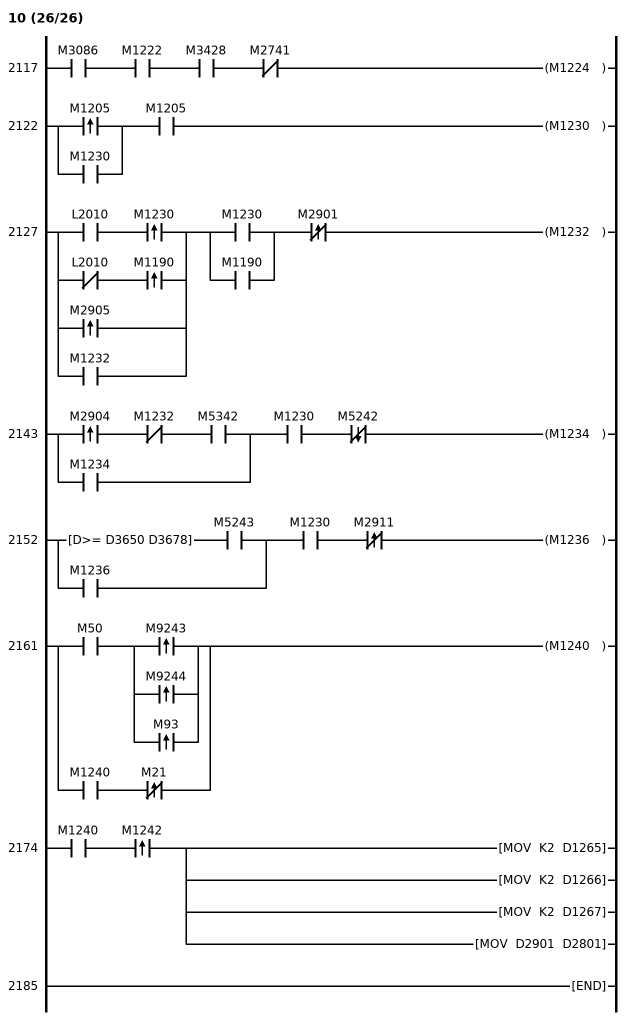
2117  LD      M3086
      AND     M1222
      AND     M3428
      ANI     M2741
      OUT     M1224
2122  LDP     M1205
      OR      M1230
      AND     M1205
      OUT     M1230
2127  LD      L2010
      ANDP    M1230
      LDI     L2010
      ANDP    M1190
      ORB
      ORP     M2905
      OR      M1232
      LD      M1230
      OR      M1190
      ANB
      ANDPI   M2901
      OUT     M1232
2143  LDP     M2904
      ANI     M1232
      AND     M5342
      OR      M1234
      AND     M1230
      ANDFI   M5242
      OUT     M1234
2152  LDD>=   D3650 D3678
      AND     M5243
      OR      M1236
      AND     M1230
      ANDPI   M2911
      OUT     M1236
2161  LD      M50
      LDP     M9243
      ORP     M9244
      ORP     M93
      ANB
      LD      M1240
      ANDPI   M21
      ORB
      OUT     M1240
2174  LD      M1240
      ANDP    M1242
      MOV     K2 D1265
      MOV     K2 D1266
      MOV     K2 D1267
      MOV     D2901 D2801
2185  END
END_PROGRAM

PROGRAM 20
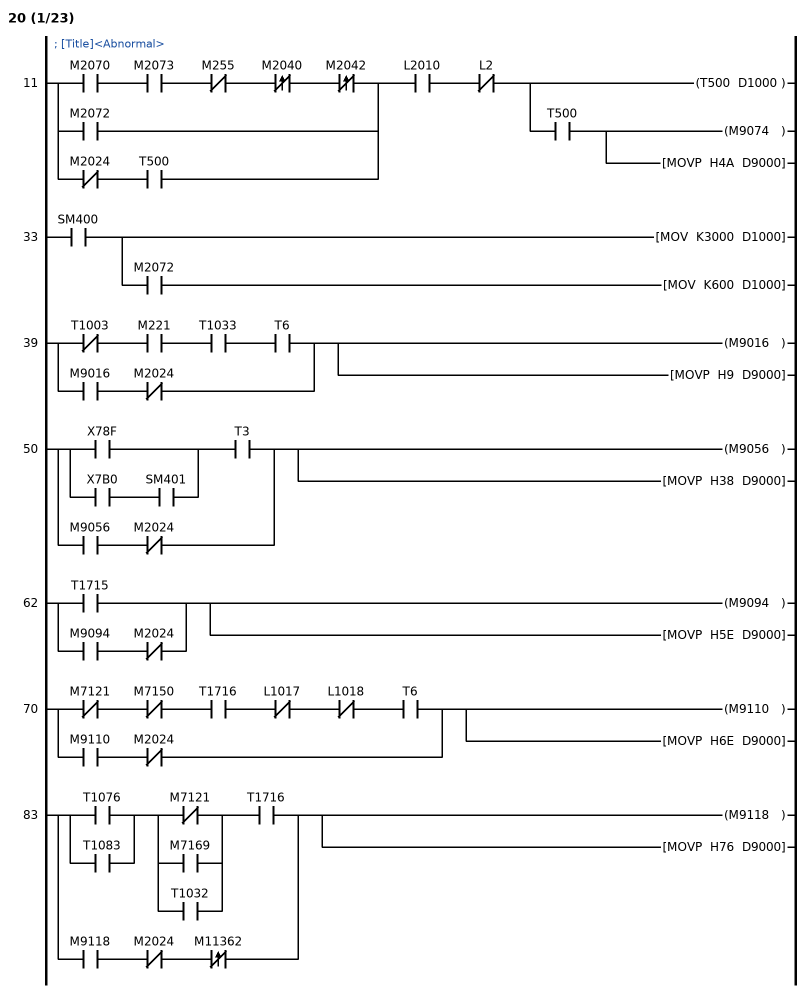
; [Title]<Abnormal>
11    LD      M2070
      AND     M2073
      ANI     M255
      ANDPI   M2040
      ANDPI   M2042
      OR      M2072
      LDI     M2024
      AND     T500
      ORB
      AND     L2010
      ANI     L2
      OUT     T500 D1000
      AND     T500
      OUT     M9074
      MOVP    H4A D9000
33    LD      SM400
      MOV     K3000 D1000
      AND     M2072
      MOV     K600 D1000
39    LDI     T1003
      AND     M221
      AND     T1033
      AND     T6
      LD      M9016
      ANI     M2024
      ORB
      OUT     M9016
      MOVP    H9 D9000
50    LD      X78F
      LD      X7B0
      AND     SM401
      ORB
      AND     T3
      LD      M9056
      ANI     M2024
      ORB
      OUT     M9056
      MOVP    H38 D9000
62    LD      T1715
      LD      M9094
      ANI     M2024
      ORB
      OUT     M9094
      MOVP    H5E D9000
70    LDI     M7121
      ANI     M7150
      AND     T1716
      ANI     L1017
      ANI     L1018
      AND     T6
      LD      M9110
      ANI     M2024
      ORB
      OUT     M9110
      MOVP    H6E D9000
83    LD      T1076
      OR      T1083
      LDI     M7121
      OR      M7169
      OR      T1032
      ANB
      AND     T1716
      LD      M9118
      ANI     M2024
      ANDPI   M11362
      ORB
      OUT     M9118
      MOVP    H76 D9000
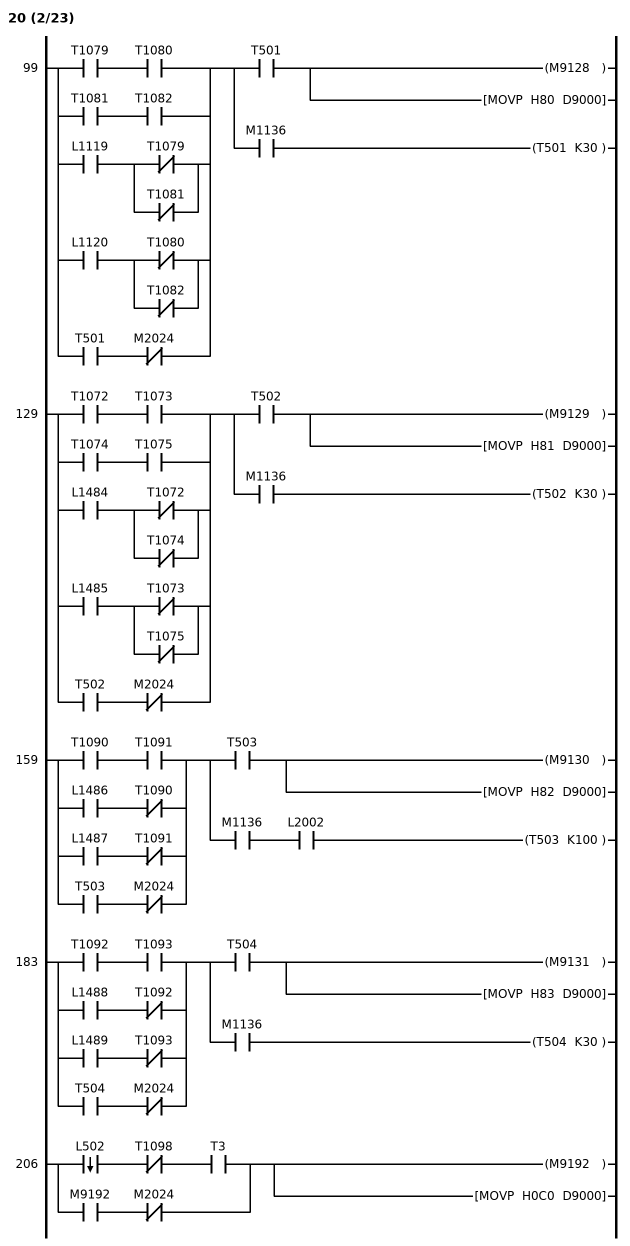
99    LD      T1079
      AND     T1080
      LD      T1081
      AND     T1082
      ORB
      LD      L1119
      LDI     T1079
      ORI     T1081
      ANB
      ORB
      LD      L1120
      LDI     T1080
      ORI     T1082
      ANB
      ORB
      LD      T501
      ANI     M2024
      ORB
      MPS
      AND     T501
      OUT     M9128
      MOVP    H80 D9000
      MPP
      AND     M1136
      OUT     T501 K30
129   LD      T1072
      AND     T1073
      LD      T1074
      AND     T1075
      ORB
      LD      L1484
      LDI     T1072
      ORI     T1074
      ANB
      ORB
      LD      L1485
      LDI     T1073
      ORI     T1075
      ANB
      ORB
      LD      T502
      ANI     M2024
      ORB
      MPS
      AND     T502
      OUT     M9129
      MOVP    H81 D9000
      MPP
      AND     M1136
      OUT     T502 K30
159   LD      T1090
      AND     T1091
      LD      L1486
      ANI     T1090
      ORB
      LD      L1487
      ANI     T1091
      ORB
      LD      T503
      ANI     M2024
      ORB
      MPS
      AND     T503
      OUT     M9130
      MOVP    H82 D9000
      MPP
      AND     M1136
      AND     L2002
      OUT     T503 K100
183   LD      T1092
      AND     T1093
      LD      L1488
      ANI     T1092
      ORB
      LD      L1489
      ANI     T1093
      ORB
      LD      T504
      ANI     M2024
      ORB
      MPS
      AND     T504
      OUT     M9131
      MOVP    H83 D9000
      MPP
      AND     M1136
      OUT     T504 K30
206   LDF     L502
      ANI     T1098
      AND     T3
      LD      M9192
      ANI     M2024
      ORB
      OUT     M9192
      MOVP    H0C0 D9000
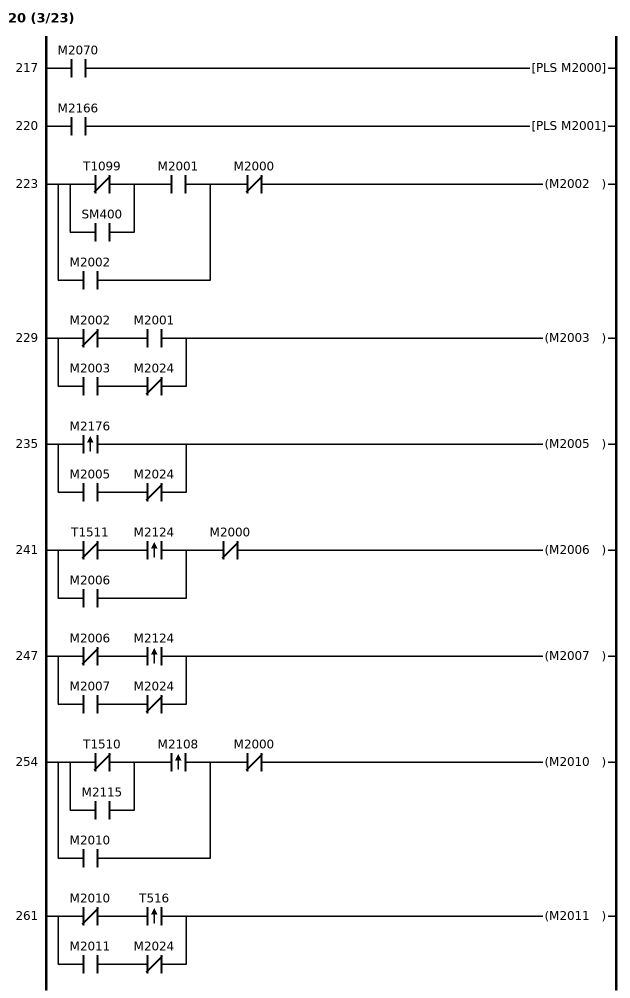
217   LD      M2070
      PLS     M2000
220   LD      M2166
      PLS     M2001
223   LDI     T1099
      OR      SM400
      AND     M2001
      OR      M2002
      ANI     M2000
      OUT     M2002
229   LDI     M2002
      AND     M2001
      LD      M2003
      ANI     M2024
      ORB
      OUT     M2003
235   LDP     M2176
      LD      M2005
      ANI     M2024
      ORB
      OUT     M2005
241   LDI     T1511
      ANDP    M2124
      OR      M2006
      ANI     M2000
      OUT     M2006
247   LDI     M2006
      ANDP    M2124
      LD      M2007
      ANI     M2024
      ORB
      OUT     M2007
254   LDI     T1510
      OR      M2115
      ANDP    M2108
      OR      M2010
      ANI     M2000
      OUT     M2010
261   LDI     M2010
      ANDP    T516
      LD      M2011
      ANI     M2024
      ORB
      OUT     M2011
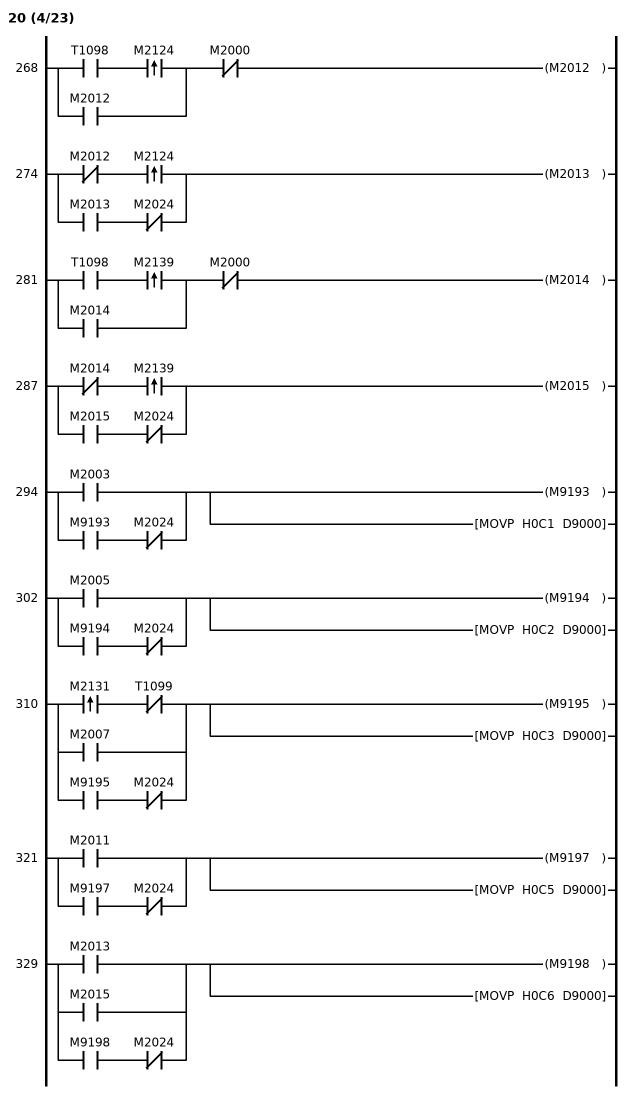
268   LD      T1098
      ANDP    M2124
      OR      M2012
      ANI     M2000
      OUT     M2012
274   LDI     M2012
      ANDP    M2124
      LD      M2013
      ANI     M2024
      ORB
      OUT     M2013
281   LD      T1098
      ANDP    M2139
      OR      M2014
      ANI     M2000
      OUT     M2014
287   LDI     M2014
      ANDP    M2139
      LD      M2015
      ANI     M2024
      ORB
      OUT     M2015
294   LD      M2003
      LD      M9193
      ANI     M2024
      ORB
      OUT     M9193
      MOVP    H0C1 D9000
302   LD      M2005
      LD      M9194
      ANI     M2024
      ORB
      OUT     M9194
      MOVP    H0C2 D9000
310   LDP     M2131
      ANI     T1099
      OR      M2007
      LD      M9195
      ANI     M2024
      ORB
      OUT     M9195
      MOVP    H0C3 D9000
321   LD      M2011
      LD      M9197
      ANI     M2024
      ORB
      OUT     M9197
      MOVP    H0C5 D9000
329   LD      M2013
      OR      M2015
      LD      M9198
      ANI     M2024
      ORB
      OUT     M9198
      MOVP    H0C6 D9000
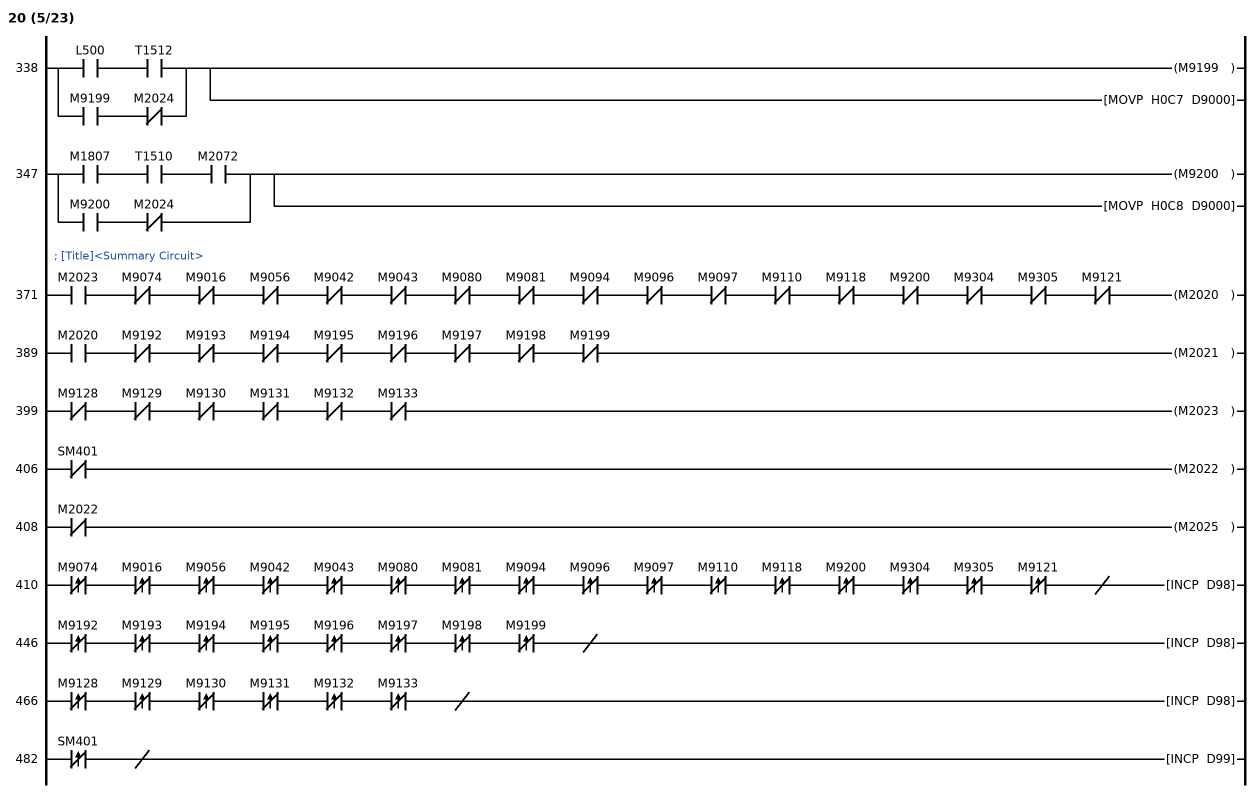
338   LD      L500
      AND     T1512
      LD      M9199
      ANI     M2024
      ORB
      OUT     M9199
      MOVP    H0C7 D9000
347   LD      M1807
      AND     T1510
      AND     M2072
      LD      M9200
      ANI     M2024
      ORB
      OUT     M9200
      MOVP    H0C8 D9000
; [Title]<Summary Circuit>
371   LD      M2023
      ANI     M9074
      ANI     M9016
      ANI     M9056
      ANI     M9042
      ANI     M9043
      ANI     M9080
      ANI     M9081
      ANI     M9094
      ANI     M9096
      ANI     M9097
      ANI     M9110
      ANI     M9118
      ANI     M9200
      ANI     M9304
      ANI     M9305
      ANI     M9121
      OUT     M2020
389   LD      M2020
      ANI     M9192
      ANI     M9193
      ANI     M9194
      ANI     M9195
      ANI     M9196
      ANI     M9197
      ANI     M9198
      ANI     M9199
      OUT     M2021
399   LDI     M9128
      ANI     M9129
      ANI     M9130
      ANI     M9131
      ANI     M9132
      ANI     M9133
      OUT     M2023
406   LDI     SM401
      OUT     M2022
408   LDI     M2022
      OUT     M2025
410   LDPI    M9074
      ANDPI   M9016
      ANDPI   M9056
      ANDPI   M9042
      ANDPI   M9043
      ANDPI   M9080
      ANDPI   M9081
      ANDPI   M9094
      ANDPI   M9096
      ANDPI   M9097
      ANDPI   M9110
      ANDPI   M9118
      ANDPI   M9200
      ANDPI   M9304
      ANDPI   M9305
      ANDPI   M9121
      INV
      INCP    D98
446   LDPI    M9192
      ANDPI   M9193
      ANDPI   M9194
      ANDPI   M9195
      ANDPI   M9196
      ANDPI   M9197
      ANDPI   M9198
      ANDPI   M9199
      INV
      INCP    D98
466   LDPI    M9128
      ANDPI   M9129
      ANDPI   M9130
      ANDPI   M9131
      ANDPI   M9132
      ANDPI   M9133
      INV
      INCP    D98
482   LDPI    SM401
      INV
      INCP    D99
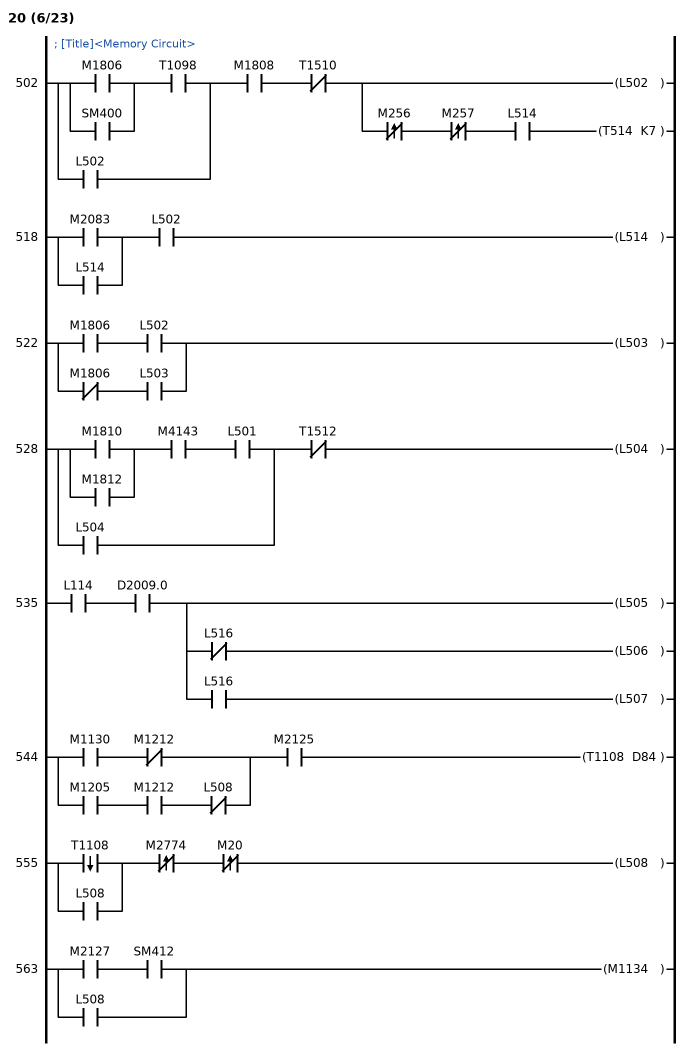
; [Title]<Memory Circuit>
502   LD      M1806
      OR      SM400
      AND     T1098
      OR      L502
      AND     M1808
      ANI     T1510
      OUT     L502
      ANDPI   M256
      ANDPI   M257
      AND     L514
      OUT     T514 K7
518   LD      M2083
      OR      L514
      AND     L502
      OUT     L514
522   LD      M1806
      AND     L502
      LDI     M1806
      AND     L503
      ORB
      OUT     L503
528   LD      M1810
      OR      M1812
      AND     M4143
      AND     L501
      OR      L504
      ANI     T1512
      OUT     L504
535   LD      L114
      AND     D2009.0
      OUT     L505
      MPS
      ANI     L516
      OUT     L506
      MPP
      AND     L516
      OUT     L507
544   LD      M1130
      ANI     M1212
      LD      M1205
      AND     M1212
      ANI     L508
      ORB
      AND     M2125
      OUT     T1108 D84
555   LDF     T1108
      OR      L508
      ANDPI   M2774
      ANDPI   M20
      OUT     L508
563   LD      M2127
      AND     SM412
      OR      L508
      OUT     M1134
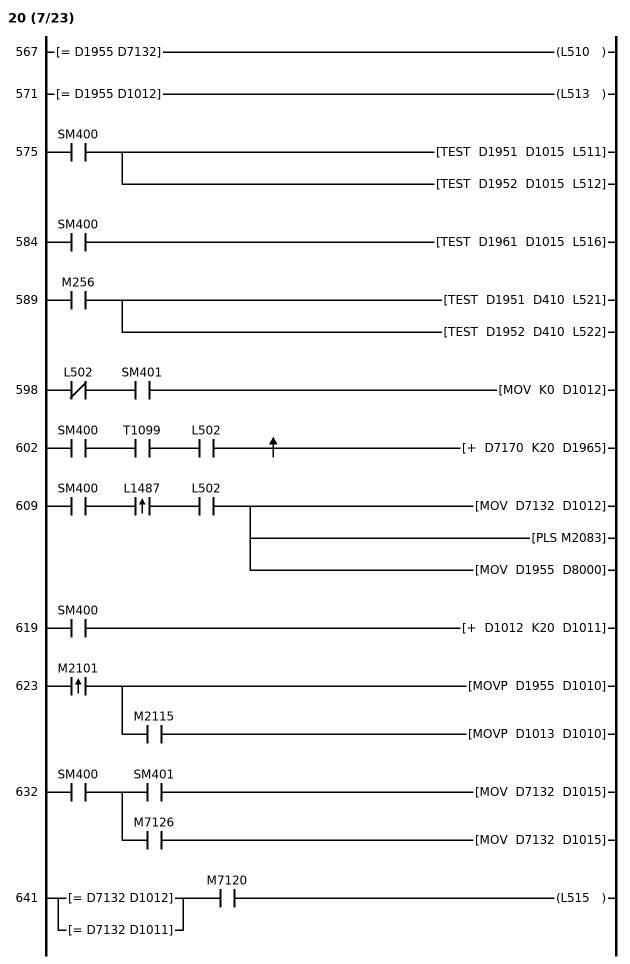
567   LD=     D1955 D7132
      OUT     L510
571   LD=     D1955 D1012
      OUT     L513
575   LD      SM400
      TEST    D1951 D1015 L511
      TEST    D1952 D1015 L512
584   LD      SM400
      TEST    D1961 D1015 L516
589   LD      M256
      TEST    D1951 D410 L521
      TEST    D1952 D410 L522
598   LDI     L502
      AND     SM401
      MOV     K0 D1012
602   LD      SM400
      AND     T1099
      AND     L502
      MEP
      +       D7170 K20 D1965
609   LD      SM400
      ANDP    L1487
      AND     L502
      MOV     D7132 D1012
      PLS     M2083
      MOV     D1955 D8000
619   LD      SM400
      +       D1012 K20 D1011
623   LDP     M2101
      MOVP    D1955 D1010
      AND     M2115
      MOVP    D1013 D1010
632   LD      SM400
      MPS
      AND     SM401
      MOV     D7132 D1015
      MPP
      AND     M7126
      MOV     D7132 D1015
641   LD=     D7132 D1012
      OR=     D7132 D1011
      AND     M7120
      OUT     L515
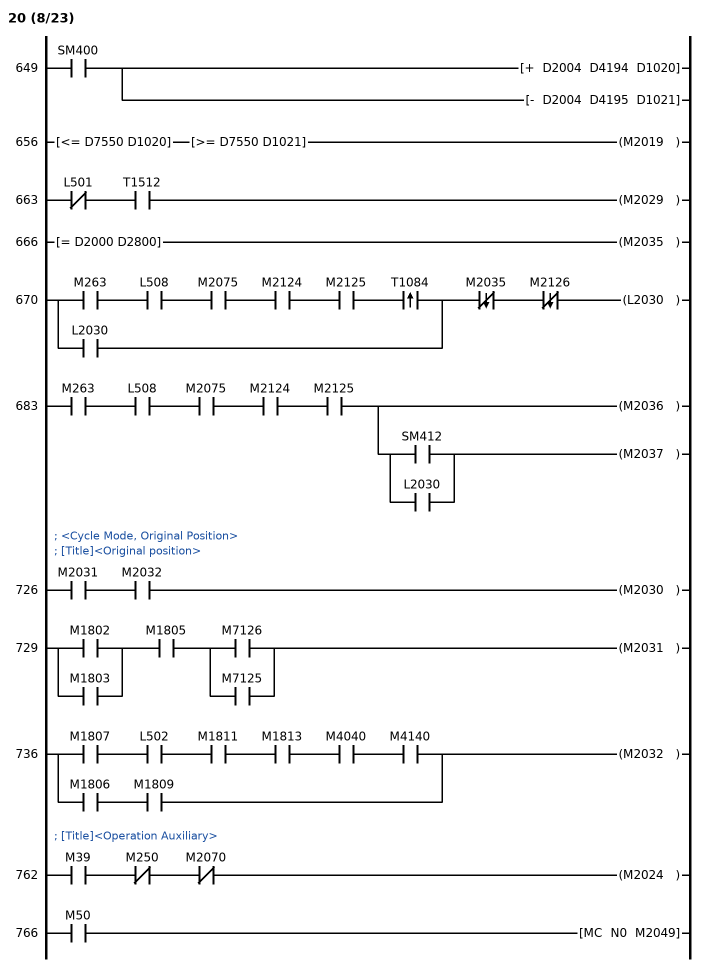
649   LD      SM400
      +       D2004 D4194 D1020
      -       D2004 D4195 D1021
656   LD<=    D7550 D1020
      AND>=   D7550 D1021
      OUT     M2019
663   LDI     L501
      AND     T1512
      OUT     M2029
666   LD=     D2000 D2800
      OUT     M2035
670   LD      M263
      AND     L508
      AND     M2075
      AND     M2124
      AND     M2125
      ANDP    T1084
      OR      L2030
      ANDFI   M2035
      ANDFI   M2126
      OUT     L2030
683   LD      M263
      AND     L508
      AND     M2075
      AND     M2124
      AND     M2125
      OUT     M2036
      LD      SM412
      OR      L2030
      ANB
      OUT     M2037
; <Cycle Mode, Original Position>
; [Title]<Original position>
726   LD      M2031
      AND     M2032
      OUT     M2030
729   LD      M1802
      OR      M1803
      AND     M1805
      LD      M7126
      OR      M7125
      ANB
      OUT     M2031
736   LD      M1807
      AND     L502
      AND     M1811
      AND     M1813
      AND     M4040
      AND     M4140
      LD      M1806
      AND     M1809
      ORB
      OUT     M2032
; [Title]<Operation Auxiliary>
762   LD      M39
      ANI     M250
      ANI     M2070
      OUT     M2024
766   LD      M50
      MC      N0 M2049
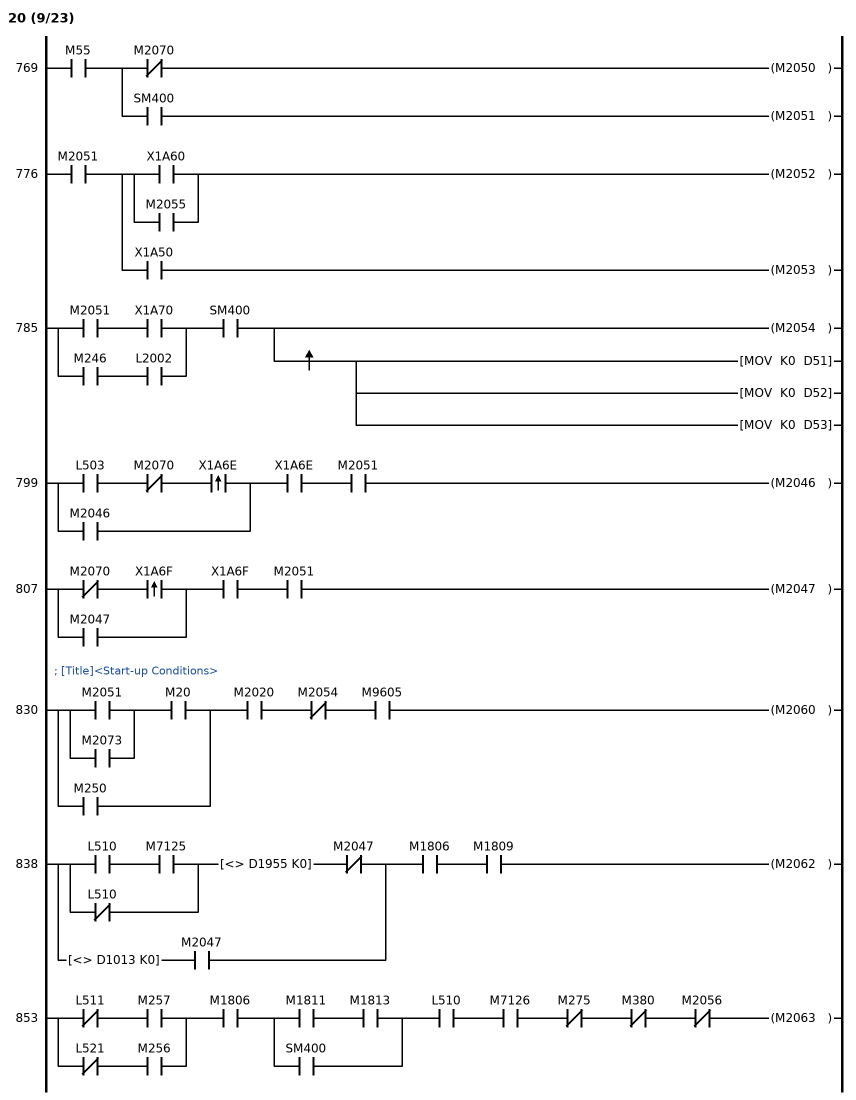
769   LD      M55
      MPS
      ANI     M2070
      OUT     M2050
      MPP
      AND     SM400
      OUT     M2051
776   LD      M2051
      MPS
      LD      X1A60
      OR      M2055
      ANB
      OUT     M2052
      MPP
      AND     X1A50
      OUT     M2053
785   LD      M2051
      AND     X1A70
      LD      M246
      AND     L2002
      ORB
      AND     SM400
      OUT     M2054
      MEP
      MOV     K0 D51
      MOV     K0 D52
      MOV     K0 D53
799   LD      L503
      ANI     M2070
      ANDP    X1A6E
      OR      M2046
      AND     X1A6E
      AND     M2051
      OUT     M2046
807   LDI     M2070
      ANDP    X1A6F
      OR      M2047
      AND     X1A6F
      AND     M2051
      OUT     M2047
; [Title]<Start-up Conditions>
830   LD      M2051
      OR      M2073
      AND     M20
      OR      M250
      AND     M2020
      ANI     M2054
      AND     M9605
      OUT     M2060
838   LD      L510
      AND     M7125
      ORI     L510
      AND<>   D1955 K0
      ANI     M2047
      LD<>    D1013 K0
      AND     M2047
      ORB
      AND     M1806
      AND     M1809
      OUT     M2062
853   LDI     L511
      AND     M257
      LDI     L521
      AND     M256
      ORB
      AND     M1806
      LD      M1811
      AND     M1813
      OR      SM400
      ANB
      AND     L510
      AND     M7126
      ANI     M275
      ANI     M380
      ANI     M2056
      OUT     M2063
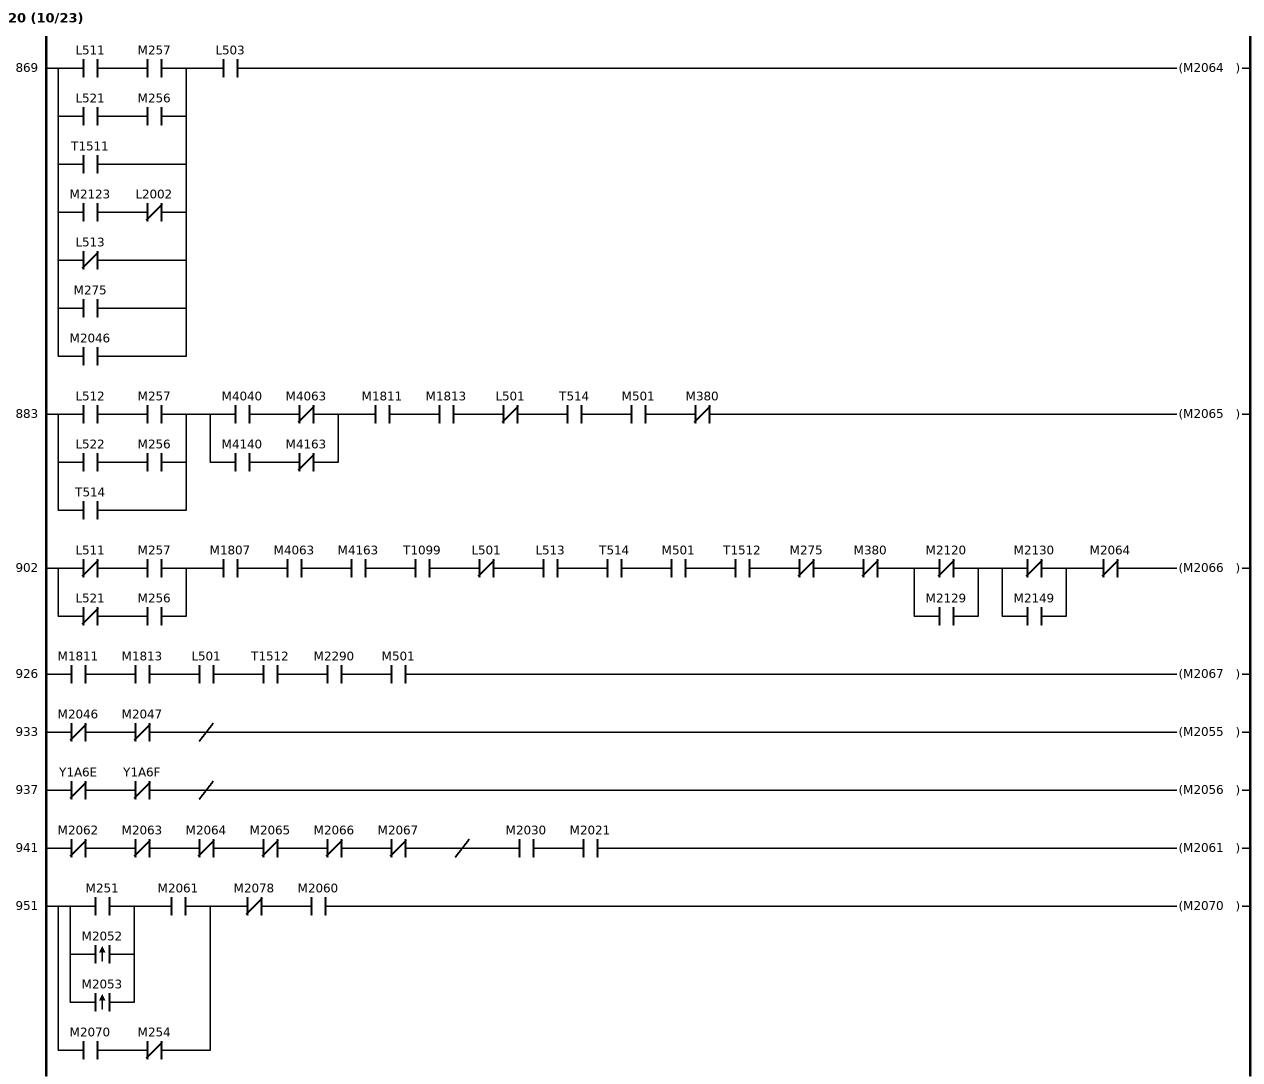
869   LD      L511
      AND     M257
      LD      L521
      AND     M256
      ORB
      OR      T1511
      LD      M2123
      ANI     L2002
      ORB
      ORI     L513
      OR      M275
      OR      M2046
      AND     L503
      OUT     M2064
883   LD      L512
      AND     M257
      LD      L522
      AND     M256
      ORB
      OR      T514
      LD      M4040
      ANI     M4063
      LD      M4140
      ANI     M4163
      ORB
      ANB
      AND     M1811
      AND     M1813
      ANI     L501
      AND     T514
      AND     M501
      ANI     M380
      OUT     M2065
902   LDI     L511
      AND     M257
      LDI     L521
      AND     M256
      ORB
      AND     M1807
      AND     M4063
      AND     M4163
      AND     T1099
      ANI     L501
      AND     L513
      AND     T514
      AND     M501
      AND     T1512
      ANI     M275
      ANI     M380
      LDI     M2120
      OR      M2129
      ANB
      LDI     M2130
      OR      M2149
      ANB
      ANI     M2064
      OUT     M2066
926   LD      M1811
      AND     M1813
      AND     L501
      AND     T1512
      AND     M2290
      AND     M501
      OUT     M2067
933   LDI     M2046
      ANI     M2047
      INV
      OUT     M2055
937   LDI     Y1A6E
      ANI     Y1A6F
      INV
      OUT     M2056
941   LDI     M2062
      ANI     M2063
      ANI     M2064
      ANI     M2065
      ANI     M2066
      ANI     M2067
      INV
      AND     M2030
      AND     M2021
      OUT     M2061
951   LD      M251
      ORP     M2052
      ORP     M2053
      AND     M2061
      LD      M2070
      ANI     M254
      ORB
      ANI     M2078
      AND     M2060
      OUT     M2070
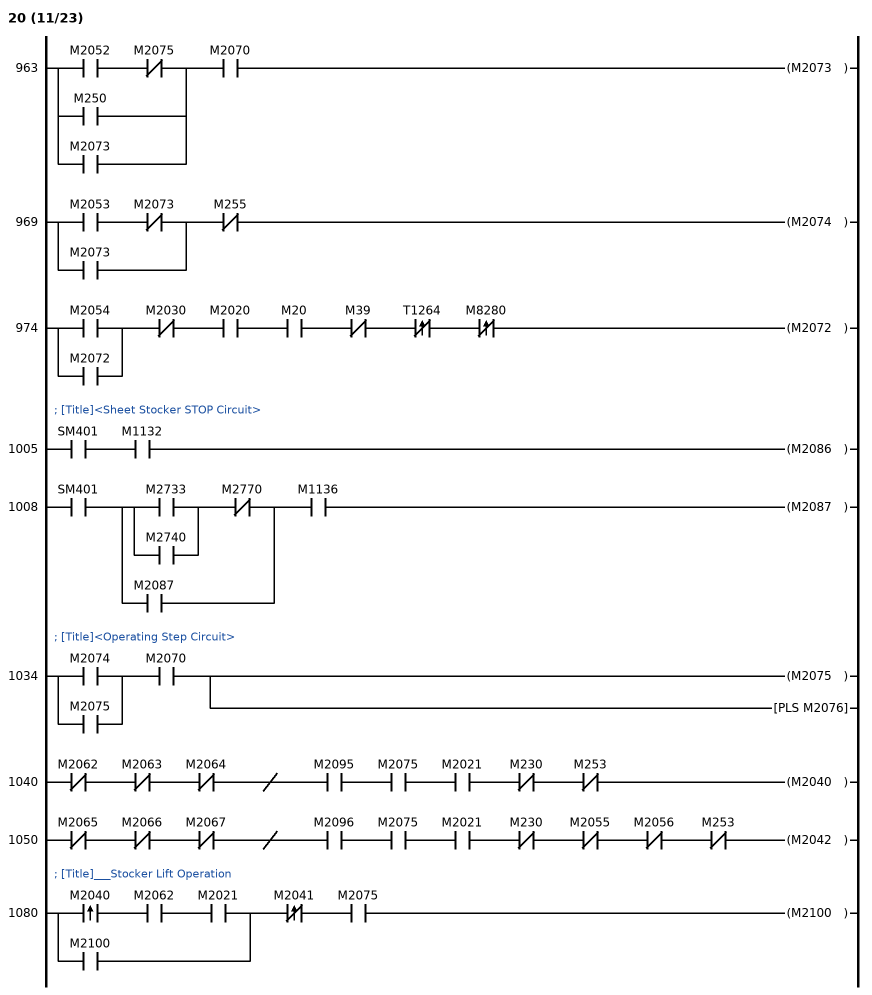
963   LD      M2052
      ANI     M2075
      OR      M250
      OR      M2073
      AND     M2070
      OUT     M2073
969   LD      M2053
      ANI     M2073
      OR      M2073
      ANI     M255
      OUT     M2074
974   LD      M2054
      OR      M2072
      ANI     M2030
      AND     M2020
      AND     M20
      ANI     M39
      ANDPI   T1264
      ANDPI   M8280
      OUT     M2072
; [Title]<Sheet Stocker STOP Circuit>
1005  LD      SM401
      AND     M1132
      OUT     M2086
1008  LD      SM401
      LD      M2733
      OR      M2740
      ANI     M2770
      OR      M2087
      ANB
      AND     M1136
      OUT     M2087
; [Title]<Operating Step Circuit>
1034  LD      M2074
      OR      M2075
      AND     M2070
      OUT     M2075
      PLS     M2076
1040  LDI     M2062
      ANI     M2063
      ANI     M2064
      INV
      AND     M2095
      AND     M2075
      AND     M2021
      ANI     M230
      ANI     M253
      OUT     M2040
1050  LDI     M2065
      ANI     M2066
      ANI     M2067
      INV
      AND     M2096
      AND     M2075
      AND     M2021
      ANI     M230
      ANI     M2055
      ANI     M2056
      ANI     M253
      OUT     M2042
; [Title]___Stocker Lift Operation
1080  LDP     M2040
      AND     M2062
      AND     M2021
      OR      M2100
      ANDPI   M2041
      AND     M2075
      OUT     M2100
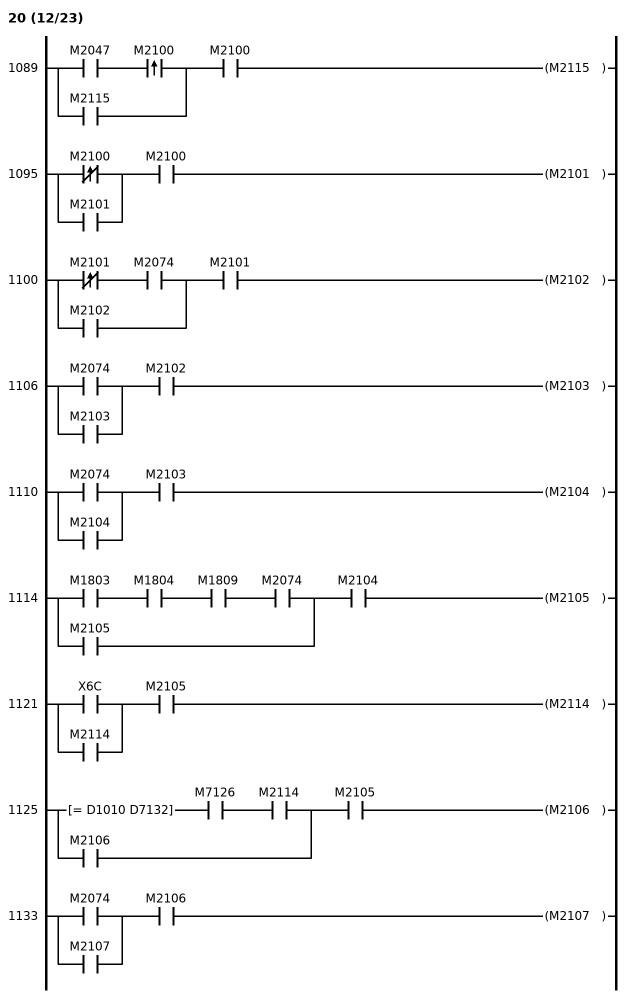
1089  LD      M2047
      ANDP    M2100
      OR      M2115
      AND     M2100
      OUT     M2115
1095  LDPI    M2100
      OR      M2101
      AND     M2100
      OUT     M2101
1100  LDPI    M2101
      AND     M2074
      OR      M2102
      AND     M2101
      OUT     M2102
1106  LD      M2074
      OR      M2103
      AND     M2102
      OUT     M2103
1110  LD      M2074
      OR      M2104
      AND     M2103
      OUT     M2104
1114  LD      M1803
      AND     M1804
      AND     M1809
      AND     M2074
      OR      M2105
      AND     M2104
      OUT     M2105
1121  LD      X6C
      OR      M2114
      AND     M2105
      OUT     M2114
1125  LD=     D1010 D7132
      AND     M7126
      AND     M2114
      OR      M2106
      AND     M2105
      OUT     M2106
1133  LD      M2074
      OR      M2107
      AND     M2106
      OUT     M2107
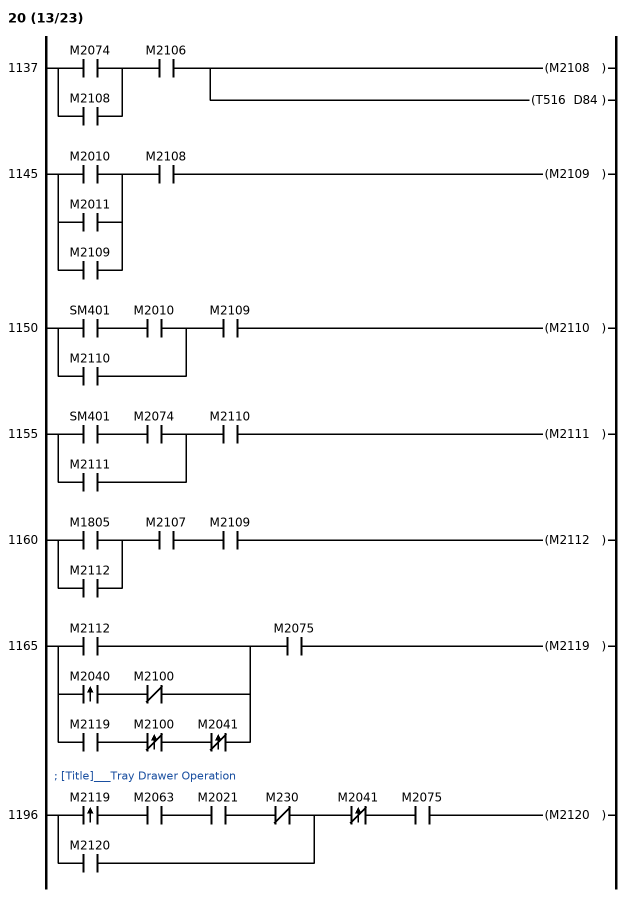
1137  LD      M2074
      OR      M2108
      AND     M2106
      OUT     M2108
      OUT     T516 D84
1145  LD      M2010
      OR      M2011
      OR      M2109
      AND     M2108
      OUT     M2109
1150  LD      SM401
      AND     M2010
      OR      M2110
      AND     M2109
      OUT     M2110
1155  LD      SM401
      AND     M2074
      OR      M2111
      AND     M2110
      OUT     M2111
1160  LD      M1805
      OR      M2112
      AND     M2107
      AND     M2109
      OUT     M2112
1165  LD      M2112
      LDP     M2040
      ANI     M2100
      ORB
      LD      M2119
      ANDPI   M2100
      ANDPI   M2041
      ORB
      AND     M2075
      OUT     M2119
; [Title]___Tray Drawer Operation
1196  LDP     M2119
      AND     M2063
      AND     M2021
      ANI     M230
      OR      M2120
      ANDPI   M2041
      AND     M2075
      OUT     M2120
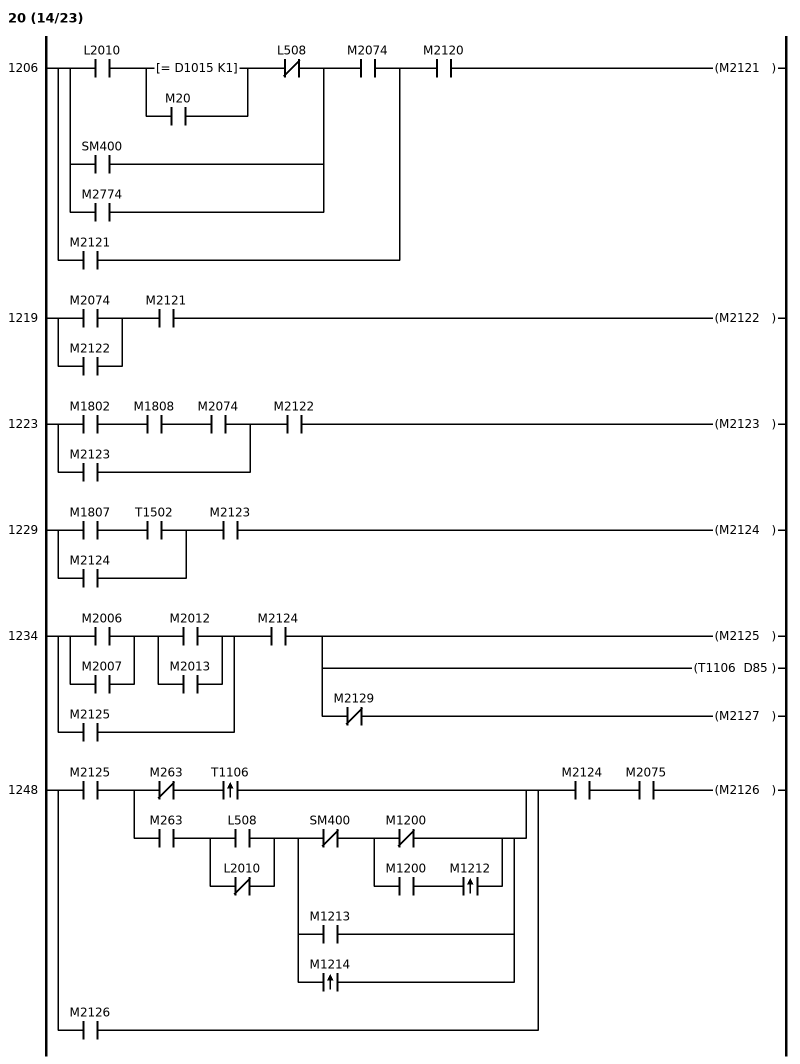
1206  LD      L2010
      LD=     D1015 K1
      OR      M20
      ANB
      ANI     L508
      OR      SM400
      OR      M2774
      AND     M2074
      OR      M2121
      AND     M2120
      OUT     M2121
1219  LD      M2074
      OR      M2122
      AND     M2121
      OUT     M2122
1223  LD      M1802
      AND     M1808
      AND     M2074
      OR      M2123
      AND     M2122
      OUT     M2123
1229  LD      M1807
      AND     T1502
      OR      M2124
      AND     M2123
      OUT     M2124
1234  LD      M2006
      OR      M2007
      LD      M2012
      OR      M2013
      ANB
      OR      M2125
      AND     M2124
      OUT     M2125
      OUT     T1106 D85
      ANI     M2129
      OUT     M2127
1248  LD      M2125
      LDI     M263
      ANDP    T1106
      LD      M263
      LD      L508
      ORI     L2010
      ANB
      LDI     SM400
      LDI     M1200
      LD      M1200
      ANDP    M1212
      ORB
      ANB
      OR      M1213
      ORP     M1214
      ANB
      ORB
      ANB
      OR      M2126
      AND     M2124
      AND     M2075
      OUT     M2126
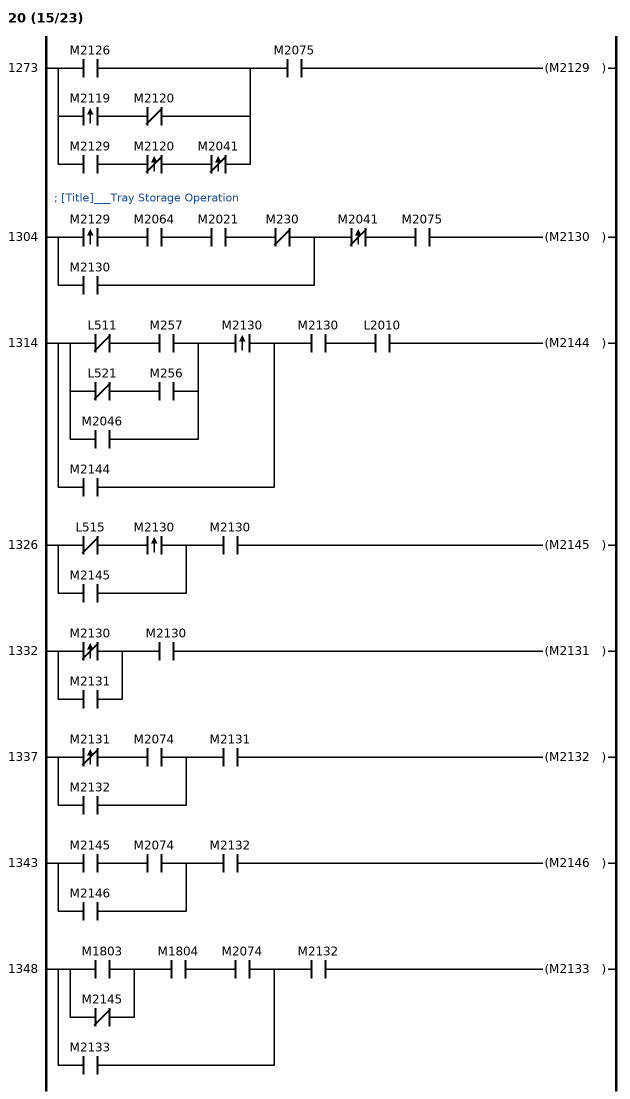
1273  LD      M2126
      LDP     M2119
      ANI     M2120
      ORB
      LD      M2129
      ANDPI   M2120
      ANDPI   M2041
      ORB
      AND     M2075
      OUT     M2129
; [Title]___Tray Storage Operation
1304  LDP     M2129
      AND     M2064
      AND     M2021
      ANI     M230
      OR      M2130
      ANDPI   M2041
      AND     M2075
      OUT     M2130
1314  LDI     L511
      AND     M257
      LDI     L521
      AND     M256
      ORB
      OR      M2046
      ANDP    M2130
      OR      M2144
      AND     M2130
      AND     L2010
      OUT     M2144
1326  LDI     L515
      ANDP    M2130
      OR      M2145
      AND     M2130
      OUT     M2145
1332  LDPI    M2130
      OR      M2131
      AND     M2130
      OUT     M2131
1337  LDPI    M2131
      AND     M2074
      OR      M2132
      AND     M2131
      OUT     M2132
1343  LD      M2145
      AND     M2074
      OR      M2146
      AND     M2132
      OUT     M2146
1348  LD      M1803
      ORI     M2145
      AND     M1804
      AND     M2074
      OR      M2133
      AND     M2132
      OUT     M2133
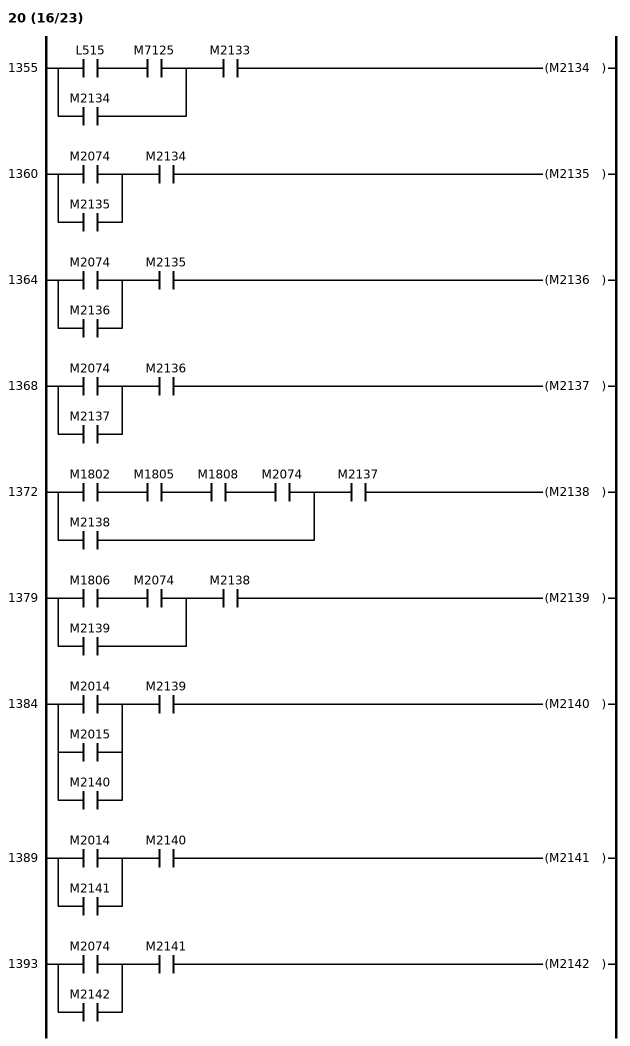
1355  LD      L515
      AND     M7125
      OR      M2134
      AND     M2133
      OUT     M2134
1360  LD      M2074
      OR      M2135
      AND     M2134
      OUT     M2135
1364  LD      M2074
      OR      M2136
      AND     M2135
      OUT     M2136
1368  LD      M2074
      OR      M2137
      AND     M2136
      OUT     M2137
1372  LD      M1802
      AND     M1805
      AND     M1808
      AND     M2074
      OR      M2138
      AND     M2137
      OUT     M2138
1379  LD      M1806
      AND     M2074
      OR      M2139
      AND     M2138
      OUT     M2139
1384  LD      M2014
      OR      M2015
      OR      M2140
      AND     M2139
      OUT     M2140
1389  LD      M2014
      OR      M2141
      AND     M2140
      OUT     M2141
1393  LD      M2074
      OR      M2142
      AND     M2141
      OUT     M2142
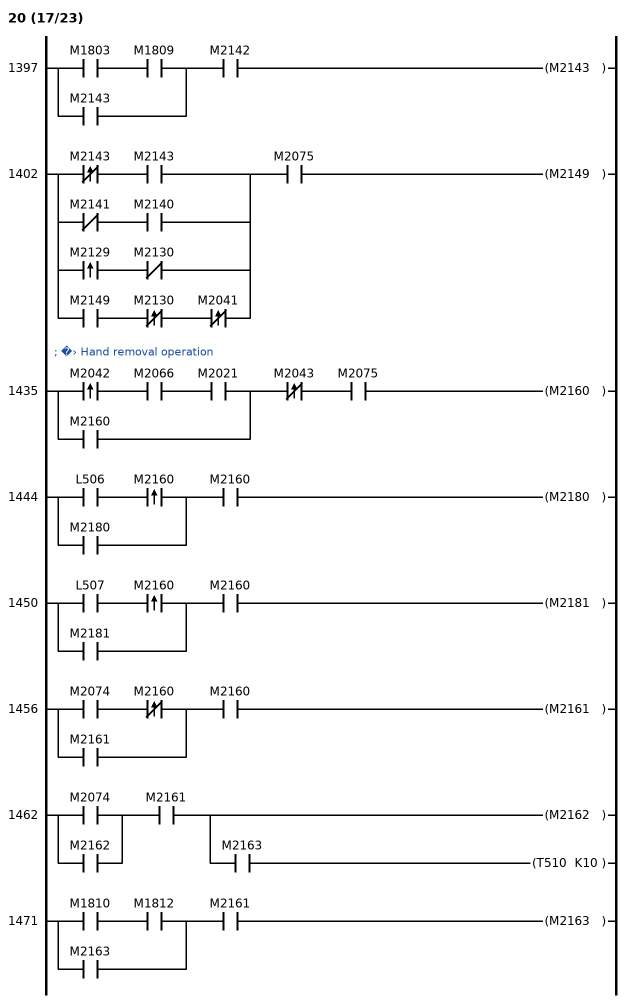
1397  LD      M1803
      AND     M1809
      OR      M2143
      AND     M2142
      OUT     M2143
1402  LDPI    M2143
      AND     M2143
      LDI     M2141
      AND     M2140
      ORB
      LDP     M2129
      ANI     M2130
      ORB
      LD      M2149
      ANDPI   M2130
      ANDPI   M2041
      ORB
      AND     M2075
      OUT     M2149
; �› Hand removal operation
1435  LDP     M2042
      AND     M2066
      AND     M2021
      OR      M2160
      ANDPI   M2043
      AND     M2075
      OUT     M2160
1444  LD      L506
      ANDP    M2160
      OR      M2180
      AND     M2160
      OUT     M2180
1450  LD      L507
      ANDP    M2160
      OR      M2181
      AND     M2160
      OUT     M2181
1456  LD      M2074
      ANDPI   M2160
      OR      M2161
      AND     M2160
      OUT     M2161
1462  LD      M2074
      OR      M2162
      AND     M2161
      OUT     M2162
      AND     M2163
      OUT     T510 K10
1471  LD      M1810
      AND     M1812
      OR      M2163
      AND     M2161
      OUT     M2163
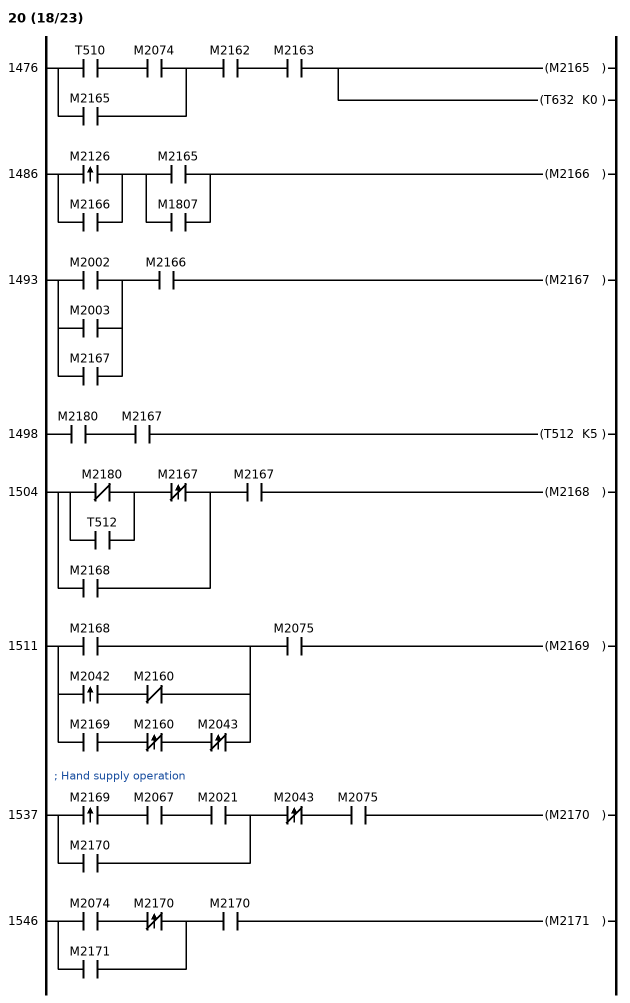
1476  LD      T510
      AND     M2074
      OR      M2165
      AND     M2162
      AND     M2163
      OUT     M2165
      OUT     T632 K0
1486  LDP     M2126
      OR      M2166
      LD      M2165
      OR      M1807
      ANB
      OUT     M2166
1493  LD      M2002
      OR      M2003
      OR      M2167
      AND     M2166
      OUT     M2167
1498  LD      M2180
      AND     M2167
      OUT     T512 K5
1504  LDI     M2180
      OR      T512
      ANDPI   M2167
      OR      M2168
      AND     M2167
      OUT     M2168
1511  LD      M2168
      LDP     M2042
      ANI     M2160
      ORB
      LD      M2169
      ANDPI   M2160
      ANDPI   M2043
      ORB
      AND     M2075
      OUT     M2169
; Hand supply operation
1537  LDP     M2169
      AND     M2067
      AND     M2021
      OR      M2170
      ANDPI   M2043
      AND     M2075
      OUT     M2170
1546  LD      M2074
      ANDPI   M2170
      OR      M2171
      AND     M2170
      OUT     M2171
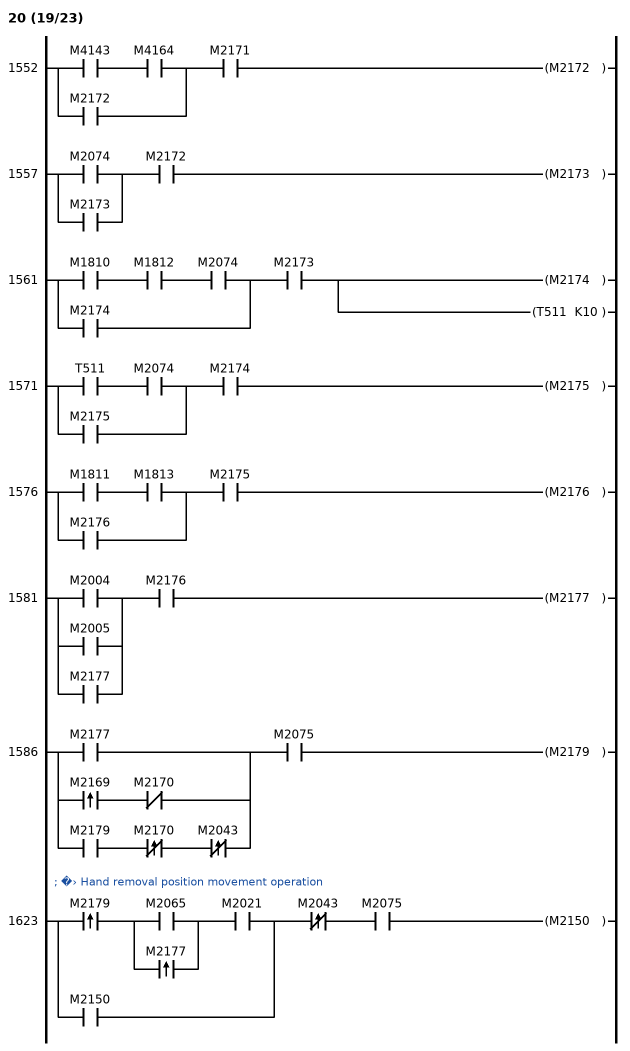
1552  LD      M4143
      AND     M4164
      OR      M2172
      AND     M2171
      OUT     M2172
1557  LD      M2074
      OR      M2173
      AND     M2172
      OUT     M2173
1561  LD      M1810
      AND     M1812
      AND     M2074
      OR      M2174
      AND     M2173
      OUT     M2174
      OUT     T511 K10
1571  LD      T511
      AND     M2074
      OR      M2175
      AND     M2174
      OUT     M2175
1576  LD      M1811
      AND     M1813
      OR      M2176
      AND     M2175
      OUT     M2176
1581  LD      M2004
      OR      M2005
      OR      M2177
      AND     M2176
      OUT     M2177
1586  LD      M2177
      LDP     M2169
      ANI     M2170
      ORB
      LD      M2179
      ANDPI   M2170
      ANDPI   M2043
      ORB
      AND     M2075
      OUT     M2179
; �› Hand removal position movement operation
1623  LDP     M2179
      LD      M2065
      ORP     M2177
      ANB
      AND     M2021
      OR      M2150
      ANDPI   M2043
      AND     M2075
      OUT     M2150
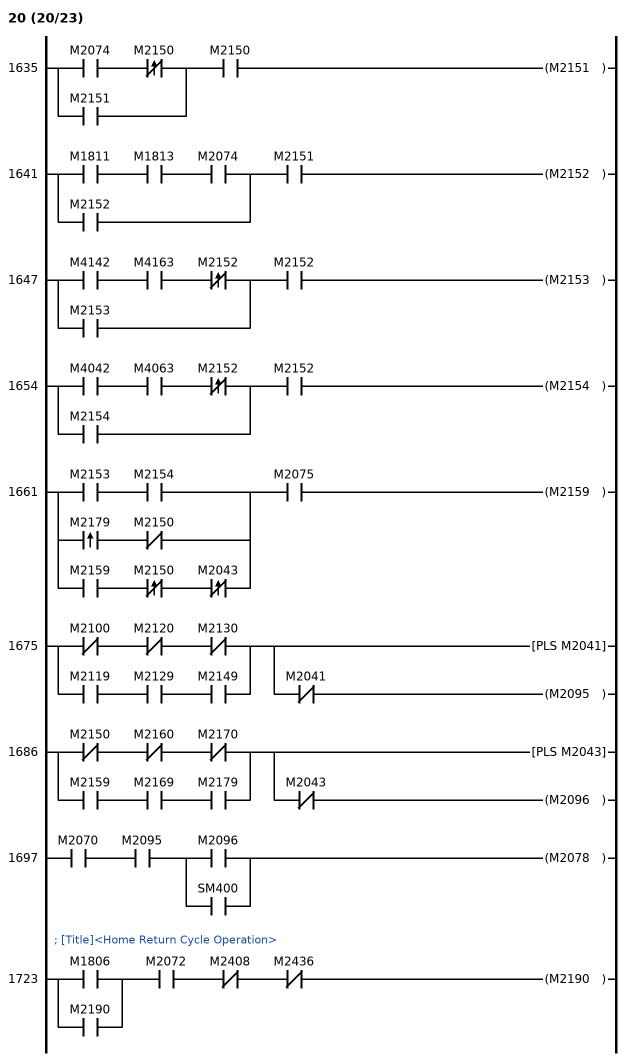
1635  LD      M2074
      ANDPI   M2150
      OR      M2151
      AND     M2150
      OUT     M2151
1641  LD      M1811
      AND     M1813
      AND     M2074
      OR      M2152
      AND     M2151
      OUT     M2152
1647  LD      M4142
      AND     M4163
      ANDPI   M2152
      OR      M2153
      AND     M2152
      OUT     M2153
1654  LD      M4042
      AND     M4063
      ANDPI   M2152
      OR      M2154
      AND     M2152
      OUT     M2154
1661  LD      M2153
      AND     M2154
      LDP     M2179
      ANI     M2150
      ORB
      LD      M2159
      ANDPI   M2150
      ANDPI   M2043
      ORB
      AND     M2075
      OUT     M2159
1675  LDI     M2100
      ANI     M2120
      ANI     M2130
      LD      M2119
      AND     M2129
      AND     M2149
      ORB
      PLS     M2041
      ANI     M2041
      OUT     M2095
1686  LDI     M2150
      ANI     M2160
      ANI     M2170
      LD      M2159
      AND     M2169
      AND     M2179
      ORB
      PLS     M2043
      ANI     M2043
      OUT     M2096
1697  LD      M2070
      AND     M2095
      LD      M2096
      OR      SM400
      ANB
      OUT     M2078
; [Title]<Home Return Cycle Operation>
1723  LD      M1806
      OR      M2190
      AND     M2072
      ANI     M2408
      ANI     M2436
      OUT     M2190
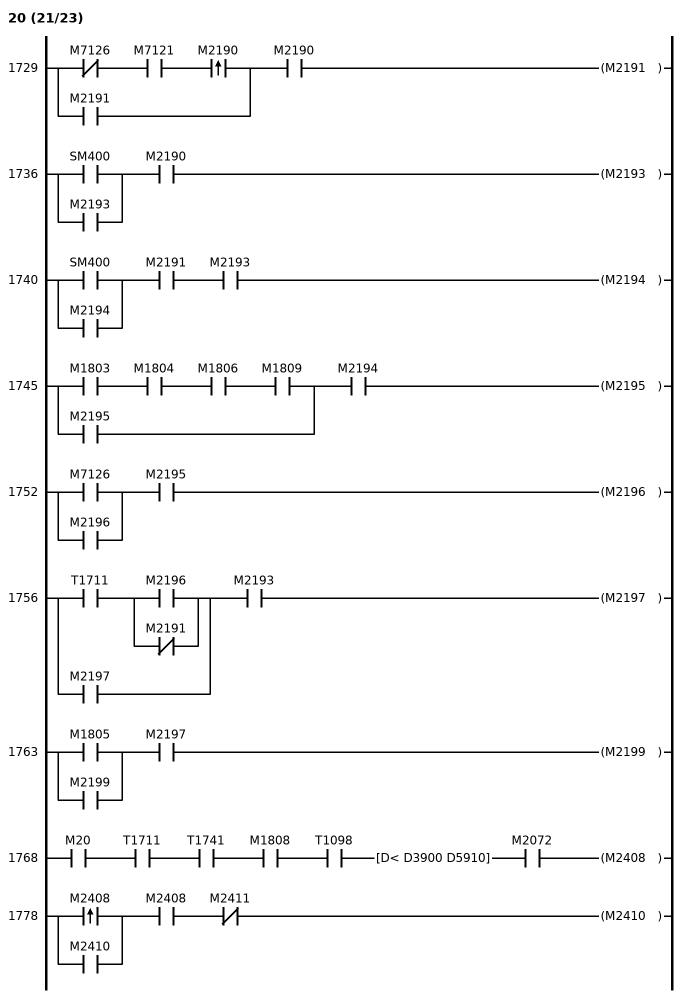
1729  LDI     M7126
      AND     M7121
      ANDP    M2190
      OR      M2191
      AND     M2190
      OUT     M2191
1736  LD      SM400
      OR      M2193
      AND     M2190
      OUT     M2193
1740  LD      SM400
      OR      M2194
      AND     M2191
      AND     M2193
      OUT     M2194
1745  LD      M1803
      AND     M1804
      AND     M1806
      AND     M1809
      OR      M2195
      AND     M2194
      OUT     M2195
1752  LD      M7126
      OR      M2196
      AND     M2195
      OUT     M2196
1756  LD      T1711
      LD      M2196
      ORI     M2191
      ANB
      OR      M2197
      AND     M2193
      OUT     M2197
1763  LD      M1805
      OR      M2199
      AND     M2197
      OUT     M2199
; 
1768  LD      M20
      AND     T1711
      AND     T1741
      AND     M1808
      AND     T1098
      ANDD<   D3900 D5910
      AND     M2072
      OUT     M2408
1778  LDP     M2408
      OR      M2410
      AND     M2408
      ANI     M2411
      OUT     M2410
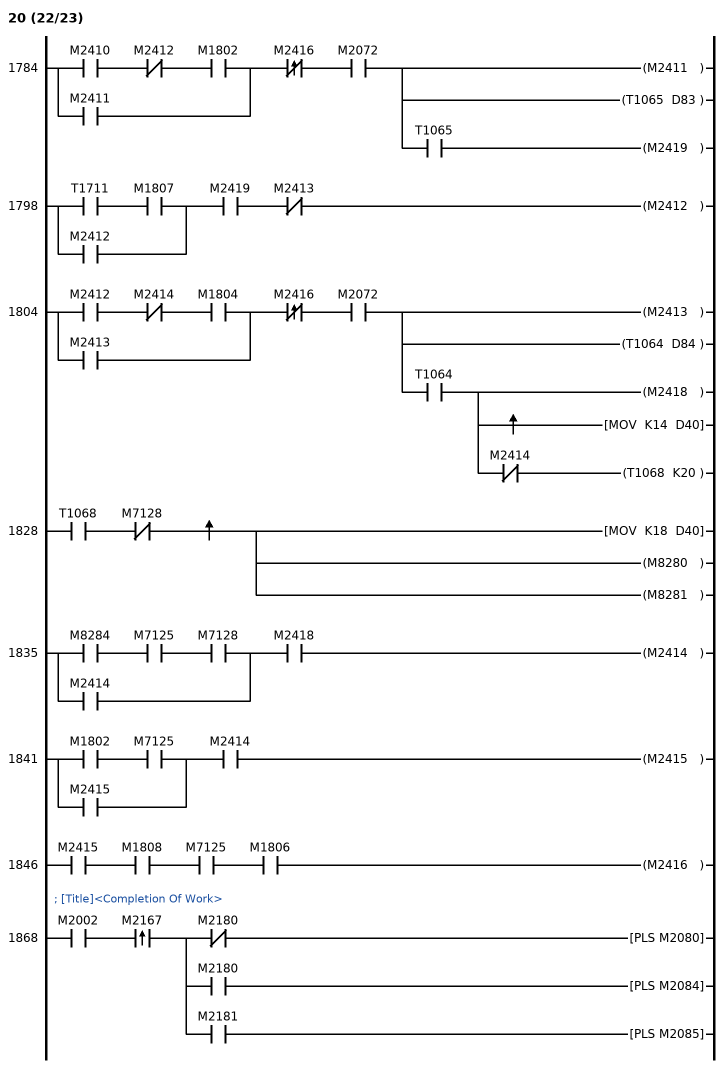
1784  LD      M2410
      ANI     M2412
      AND     M1802
      OR      M2411
      ANDPI   M2416
      AND     M2072
      OUT     M2411
      OUT     T1065 D83
      AND     T1065
      OUT     M2419
1798  LD      T1711
      AND     M1807
      OR      M2412
      AND     M2419
      ANI     M2413
      OUT     M2412
1804  LD      M2412
      ANI     M2414
      AND     M1804
      OR      M2413
      ANDPI   M2416
      AND     M2072
      OUT     M2413
      OUT     T1064 D84
      AND     T1064
      OUT     M2418
      MPS
      MEP
      MOV     K14 D40
      MPP
      ANI     M2414
      OUT     T1068 K20
1828  LD      T1068
      ANI     M7128
      MEP
      MOV     K18 D40
      OUT     M8280
      OUT     M8281
1835  LD      M8284
      AND     M7125
      AND     M7128
      OR      M2414
      AND     M2418
      OUT     M2414
1841  LD      M1802
      AND     M7125
      OR      M2415
      AND     M2414
      OUT     M2415
1846  LD      M2415
      AND     M1808
      AND     M7125
      AND     M1806
      OUT     M2416
; 
; [Title]<Completion Of Work>
1868  LD      M2002
      ANDP    M2167
      MPS
      ANI     M2180
      PLS     M2080
      MRD
      AND     M2180
      PLS     M2084
      MPP
      AND     M2181
      PLS     M2085
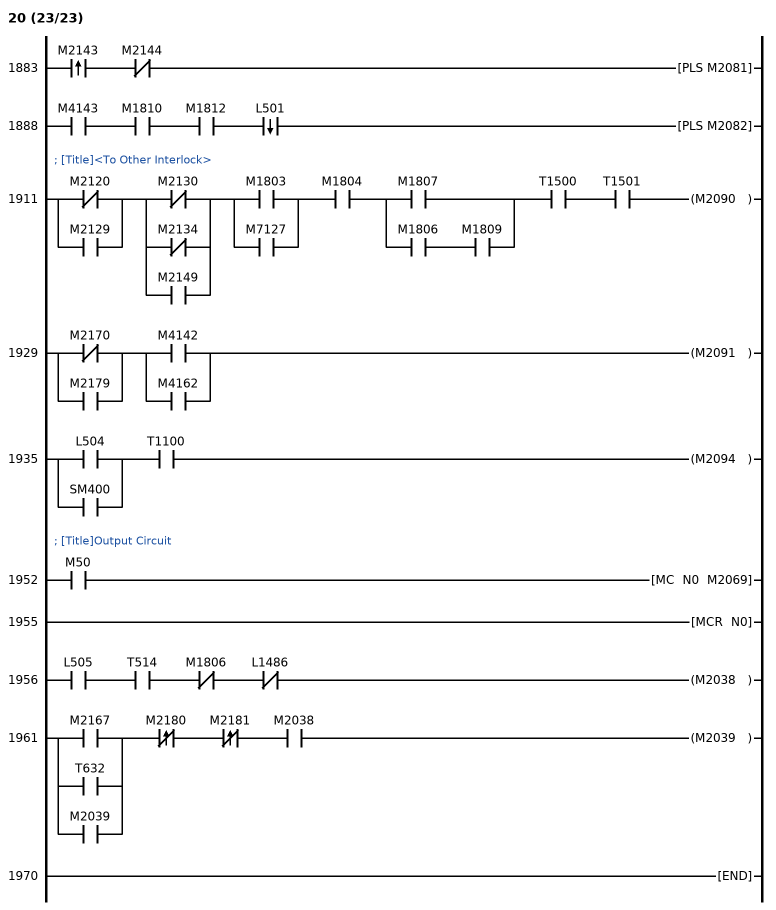
1883  LDP     M2143
      ANI     M2144
      PLS     M2081
1888  LD      M4143
      AND     M1810
      AND     M1812
      ANDF    L501
      PLS     M2082
; [Title]<To Other Interlock>
1911  LDI     M2120
      OR      M2129
      LDI     M2130
      ORI     M2134
      OR      M2149
      ANB
      LD      M1803
      OR      M7127
      ANB
      AND     M1804
      LD      M1807
      LD      M1806
      AND     M1809
      ORB
      ANB
      AND     T1500
      AND     T1501
      OUT     M2090
1929  LDI     M2170
      OR      M2179
      LD      M4142
      OR      M4162
      ANB
      OUT     M2091
1935  LD      L504
      OR      SM400
      AND     T1100
      OUT     M2094
; [Title]Output Circuit
1952  LD      M50
      MC      N0 M2069
1955  MCR     N0
1956  LD      L505
      AND     T514
      ANI     M1806
      ANI     L1486
      OUT     M2038
1961  LD      M2167
      OR      T632
      OR      M2039
      ANDPI   M2180
      ANDPI   M2181
      AND     M2038
      OUT     M2039
1970  END
END_PROGRAM

PROGRAM 21
